// TIA Portal V21 export
// export: Created 2000-01-01T00:00:00.0000000Z, ExportSetting None
FUNCTION "FC_StartStop" : Void   // FC10, SCL
{ S7_Optimized_Access := 'TRUE' }
// 起保停（Start-Hold-Stop）功能：通过全局 PLC 变量 I_Start / I_Stop / I_EStop 输入，
// 锁存输出 Q_Run。优先级：急停 > 停止 > 启动。
// 全局变量在 DefaultTagTable 中定义；HMI 通过 SetBit/ResetBit 写 I_Start/I_Stop。
// stored: SetENOAutomatically false
BEGIN
// 起保停核心逻辑
// 读全局输入 I_EStop / I_Stop / I_Start，写全局输出 Q_Run（锁存）
   IF "I_EStop" THEN
     "Q_Run" := FALSE;
   ELSIF "I_Stop" THEN
     "Q_Run" := FALSE;
   ELSIF "I_Start" THEN
     "Q_Run" := TRUE;
   END_IF;
END_FUNCTION
